FUNCTION_BLOCK FB_EventSubscriber1 IMPLEMENTS I_Observer
VAR_INPUT
	eventPublisher					: I_EventPublisher;
END_VAR
VAR
	_verbose						: BOOL := TRUE;
	_event							: INT;
	// Register after online change 
	registeredAtPublisher			: BOOL;
END_VAR

// Is there a valid publisher attached? 
IF eventPublisher=0	THEN
	RETURN;
END_IF

// Did we already register in the publisher?
IF NOT registeredAtPublisher	THEN
	registeredAtPublisher := eventPublisher.attach(THIS^);
END_IF

METHOD INTERNAL message : BOOL
VAR_INPUT
	dintArg						: DINT;
END_VAR
// Log message
IF _verbose  THEN
	ADSLOGDINT(
		msgCtrlMask := ADSLOG_MSGTYPE_HINT OR ADSLOG_MSGTYPE_LOG, // ADSLOG_MSGTYPE_ERROR OR ADSLOG_MSGTYPE_LOG, 
		msgFmtStr 	:= 'Subscriber 1 knows the value changed to %d',
		dintArg 	:= dintArg
		);
END_IF
END_METHOD

METHOD update : BOOL
// the publisher mentions an update, fetch the data
_event := eventPublisher.event;
message(TO_DINT(_event));
END_METHOD

END_FUNCTION_BLOCK

(* stored: Version 1.1.0.1, ProductVersion 3.1.4024.11
   POU FB_EventSubscriber1: Id {d4dce0f2-3ded-43b2-8491-9014ab19c774}, SpecialFunc None
   Method message: Id {e4f26ffc-57fb-4c96-b5ee-4b9c9356b25c}
   Method update: Id {26657e55-00fd-4c13-80e1-21813364b2ff} *)
